(* IEC 61131-3 sources: repolevel_ST_code_completion/dataset/project_code/traffic_light/FUN, 3 files *)

(* ---- F_SecondsToTime.st ---- *)
FUNCTION F_SecondsToTime : TIME
VAR_INPUT
	dwSeconds	:	DWORD;		//输入的秒数
END_VAR

// 将秒数（DWORD）转换为TIME类型
// 秒数乘以1000得到毫秒
F_SecondsToTime := DWORD_TO_TIME(dwSeconds * 1000);

(* ---- F_TimeToSeconds.st ---- *)
FUNCTION F_TimeToSeconds : DWORD
VAR_INPUT
	tTime	:	TIME;		//输入的时间
END_VAR

// 将TIME类型转换为秒数（DWORD）
// TIME内部是毫秒，除以1000得到秒数
F_TimeToSeconds := DINT_TO_DWORD(TRUNC(TIME_TO_DWORD(tTime) / 1000.0));

(* ---- FB_CountdownTimer.st ---- *)
FUNCTION_BLOCK FB_CountdownTimer
VAR_INPUT
	tElapsedTime	:	TIME;		//已经过的时间（定时器的ET）
	tTotalTime		:	TIME;		//总时间（定时器的PT）
END_VAR
VAR_OUTPUT
	nRemainingSeconds	:	UINT;	//剩余秒数
END_VAR
VAR
	nTotalSeconds		:	UINT;	//总秒数
	nElapsedSeconds		:	UINT;	//已过秒数
END_VAR

// 将TIME转换为秒
nTotalSeconds := INT_TO_USINT(TRUNC_INT(TIME_TO_DWORD(tTotalTime) / 1000.0));
nElapsedSeconds := INT_TO_USINT(TRUNC_INT(TIME_TO_UINT(tElapsedTime) / 1000.0));

// 计算剩余秒数
nRemainingSeconds := nTotalSeconds - nElapsedSeconds;
